TEXTLIST Seq_list
  0 = 'CYCLE START'
  10 = 'ROLLER DOOR_CLOSE'
  20 = 'TRUNION ROTATES -20*'
  30 = 'ROLLER DOOR OPEN'
  40 = 'OPERATOR LOAD 1st PART'
  50 = 'OPERATOR LOAD 2nd PART'
  60 = '1st, 3rd & 5th CLAMP CLOSE'
  70 = 'ROLLER DOOR_CLOSE'
  80 = 'TRUNION ROTATES 80*'
  90 = 'ROLLER DOOR OPEN'
  100 = 'OPERATOR LOAD_3rd_PART'
  110 = 'OPERATOR LOAD_4th_PART'
  120 = 'ROLLER DOOR_CLOSE'
  130 = '2nd, 4th & 6th CLAMP CLOSE'
  140 = 'TURNTABLE-180* AND TRUNION-0*'
  150 = 'Start WELD_Robot FOR WELD'
  160 = '1st, 3rd & 5th UNCLAMP'
  170 = 'ROLLER DOOR OPEN'
  180 = 'Start MH_Robot_1ST TIME'
  190 = 'TRUNION ROTATES 45*'
  200 = '2nd, 4th & 6th UNCLAMP '
  210 = 'Start MH_Robot_2ND TIME'
  220 = 'CYCLE COMPLETE'
  5 = 'WAIT FOR STATION HOME'
   = ''
END_TEXTLIST

(* stored: Version 1.1.0.1, ProductVersion 3.1.4024.16
   TextList Seq_list: Id {5fb94b9e-8a1a-427b-be9e-ac42e447a106} *)
